// TIA Portal V19 export
TYPE "SpeedMotor_Config"
// stored: Access Published
   STRUCT
      ReferenceVelocity : LReal;   // Reference velocity of sinamcs drive (rpm)
      InvertDirection : Bool;   // Invert direction of axis
   END_STRUCT;
END_TYPE
